// TIA Portal V18 export
DATA_BLOCK "HC1_PID_3Step"   // DB1072
// stored: AutoNumber false, DBAccessibleFromOPCUA true, InstanceOfName PID_3Step, OfSystemLibElement PID_3Step, OfSystemLibVersion 2.3
PID_3Step   // technology object, version 2.3
   // VAR_INPUT
   //    Setpoint : Real;
   //    Input : Real;
   //    Input_PER : Int;
   //    Actuator_H : Bool;
   //    Actuator_L : Bool;
   //    Feedback : Real;
   //    Feedback_PER : Int;
   //    Disturbance : Real;
   //    ManualEnable : Bool;
   //    ManualValue : Real;
   //    Manual_UP : Bool;
   //    Manual_DN : Bool;
   //    ErrorAck : Bool;
   //    Reset : Bool;
   //    ModeActivate : Bool;
   // END_VAR
   // VAR_OUTPUT
   //    ScaledInput { ExternalWritable := 'False'} : Real;
   //    ScaledFeedback { ExternalWritable := 'False'} : Real;
   //    Output_UP { ExternalWritable := 'False'} : Bool;
   //    Output_DN { ExternalWritable := 'False'} : Bool;
   //    Output_PER { ExternalWritable := 'False'} : Int;
   //    SetpointLimit_H { ExternalWritable := 'False'} : Bool;
   //    SetpointLimit_L { ExternalWritable := 'False'} : Bool;
   //    InputWarning_H { ExternalWritable := 'False'} : Bool;
   //    InputWarning_L { ExternalWritable := 'False'} : Bool;
   //    State { ExternalWritable := 'False'} : Int;
   //    Error { ExternalWritable := 'False'} : Bool;
   //    ErrorBits { ExternalWritable := 'False'} : DWord;
   // END_VAR
   // VAR_IN_OUT
   //    Mode : Int := 3;
   // END_VAR
   // VAR
   //    InternalDiagnostic : DWord;
   //    InternalVersion { ExternalWritable := 'False'} : DWord;
   //    InternalRTVersion : DWord;
   //    ManualUpInternal : Bool;
   //    ManualDnInternal : Bool;
   //    ActivateRecoverMode { S7_SetPoint := 'True'} : Bool;
   //    RunModeByStartup { S7_SetPoint := 'True'} : Bool;
   //    LoadBackUp : Bool;
   //    PhysicalUnit { ExternalWritable := 'False'; S7_SetPoint := 'True'} : Int;
   //    PhysicalQuantity { ExternalWritable := 'False'; S7_SetPoint := 'True'} : Int := 1;
   //    ErrorBehaviour { S7_SetPoint := 'True'} : Bool;
   // END_VAR
   // VAR RETAIN
   //    Warning { ExternalWritable := 'False'} : DWord;
   //    WarningInternal { ExternalWritable := 'False'} : DWord;
   // END_VAR
   // VAR
   //    SavePosition { S7_SetPoint := 'True'} : Real;
   //    CurrentSetpoint { ExternalWritable := 'False'} : Real;
   //    CancelTuningLevel { S7_SetPoint := 'True'} : Real;
   //    Progress { ExternalWritable := 'False'} : Real;
   //    Config { S7_SetPoint := 'True'} : PID_3StepConfig;
   //    GetTransitTime { S7_SetPoint := 'True'} : PID_3StepGetTransitTime;
   //    CycleTime { S7_SetPoint := 'True'} : PID_CycleTime;
   //    CtrlParamsBackUp { S7_SetPoint := 'True'} : PID_3StepControlParams;
   //    PIDSelfTune { S7_SetPoint := 'True'} : PID_3StepSelfTune;
   // END_VAR
   // VAR RETAIN
   //    Retain { S7_SetPoint := 'True'} : PID_3StepRetain;
   // END_VAR
BEGIN
   Config.InputPerOn := FALSE;
   Config.OutputPerOn := FALSE;
   Config.InputUpperLimit := 90.0;
   Config.InputLowerLimit := 15.0;
   Retain.TransitTime := 135.0;
   Retain.CtrlParams.SetByUser := TRUE;
END_DATA_BLOCK
